Staubli VAL3: cognexComm.dtx

num coGF = 10
num coGV = 1
num coLF = 9
num coLO = 8
num coSE = 7
num coSF = 4
num coSI = 3
num coSO = 2
num coSS = 5
num coSW = 6
num coTF = 11
num errorCode[10]
  [0] = 1
  [1] = 1
num nCommand[10]
  [1] = 1
num nHandleCount = 1
string strVersion = "0.3"
string tabGF[10]
  [0] = "Unrecognized command"
  [2] = "The active job has not been saved"
  [9] = "Communication Error"
string tabGV[10]
  [0] = "Unrecognized command"
  [1] = "Invalid Cell ID"
  [2] = "Command could not be executed"
  [3] = "Could not convert to num"
  [4] = "Wrong cell format : "
  [9] = "Communication Error"
string tabLF[10]
  [0] = "Unrecognized command"
  [1] = "The filename is missing"
  [2] = "The job failed to load, the system is online, or the file was not found"
  [4] = "The job to be loaded was not found, or the processor is out of memory"
  [6] = "User does not have Full Access to execute the command"
  [9] = "Communication Error"
string tabLO[10]
  [0] = "Unrecognized command"
  [1] = "Wrong user name or password"
  [9] = "Communication Error"
string tabSE[10]
  [0] = "Unrecognized command"
  [1] = "Parameter is out of range"
  [2] = "Could not execute command or system is offline"
  [9] = "Communication Error"
string tabSF[10]
  [0] = "Unrecognized command"
  [1] = "Invalid Cell ID"
  [2] = "Could not execute command or parameter out of range"
  [9] = "Communication Error"
string tabSI[10]
  [0] = "Unrecognized Command"
  [1] = "Invalid Cell ID"
  [2] = "Could not execute command or parameter is out of range"
  [9] = "Communication Error"
string tabSO[10]
  [0] = "Unrecognized command"
  [1] = "Parameter is out of range or not a valid integer"
  [5] = "Could not set online because system is set offline manually"
  [9] = "Communication Error"
string tabSS[10]
  [0] = "Unrecognized Command"
  [1] = "Invalid Cell ID"
  [5] = "The input string is too long for EditString function"
  [9] = "Communication Error"
string tabSW[10]
  [0] = "Unrecognized command"
  [1] = "Parameter is out of range"
  [2] = "Could not execute command or system is offline"
  [9] = "Communication Error"
string tabTF[10]
  [0] = "Unrecognized command"
  [1] = "The filename is missing"
  [2] = "The job failed to save, the system is online or the file was not found"
  [6] = "User does not have Full Access to execute the command"
  [9] = "Communication Error"
public bool bDebug
sio sSocket[10]
sio skCamera = {link=Socket\cognex1}
